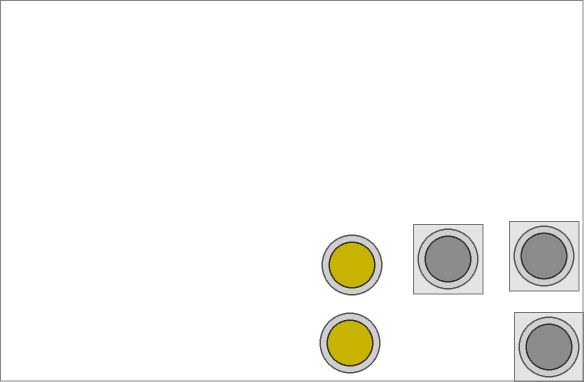
VISUALIZATION Visualization  // 584x382
    Lamp1 (317,230 70x70), variable: MAIN.bLed1, style: Lamp-Lamp1-Yellow
    Lamp1 (315,308 70x70), variable: MAIN.bLED2, style: Lamp-Lamp1-Yellow
    PushSwitch (413,224 70x70), variable: MAIN.BButton1, behaviour: TAP, style: Switch-PushSwitch-Gray
    PushSwitch (509,221 70x70), variable: MAIN.bButton2, behaviour: TAP, style: Switch-PushSwitch-Gray
    PushSwitch (514,312 70x70), variable: MAIN.bButton3, behaviour: TAP, style: Switch-PushSwitch-Gray
END_VISUALIZATION

(* stored: Version 1.1.0.1, ProductVersion 3.1.4024.12
   Visu Visualization: Id {248792c5-f220-491a-be8f-30638582143c} *)
